"H0CRM1"	Q 662.0	BOOL	// [H0IM2.H0S21]: H0: COMANDO RECUO MOTOR M1
"H0CAM1"	Q 662.1	BOOL	// [H0IM2.H0S21]: H0: COMANDO AVANÇO MOTOR M1
"H0EAPLA"	Q 700.0	BOOL	// [H0DTS1]: H0: EV RETROCESO PILOTO A
"H0ERPLA"	Q 700.1	BOOL	// [H0DTS1]: H0: EV AVANCE PILOTO A
"H0EASRB"	Q 700.2	BOOL	// [H0DTS1]: H0: EV RETROCESO SERRAGE B
"H0ERSRB"	Q 700.3	BOOL	// [H0DTS1]: H0: EV AVANCE SERRAGE B
"H0EASRC"	Q 700.4	BOOL	// [H0DTS1]: H0: EV RETROCESO SERRAGE C
"H0ERSRC"	Q 700.5	BOOL	// [H0DTS1]: H0: EV AVANCE SERRAGE C
"H0EASRD"	Q 700.6	BOOL	// [H0DTS1]: H0: EV RETROCESO SERRAGE D
"H0ERSRD"	Q 700.7	BOOL	// [H0DTS1]: H0: EV AVANCE SERRAGE D
"H0EASRE"	Q 701.0	BOOL	// [H0DTS1]: H0: EV RETROCESO SERRAGE E
"H0ERSRE"	Q 701.1	BOOL	// [H0DTS1]: H0: EV AVANCE SERRAGE E
"H0EASRF"	Q 701.2	BOOL	// [H0DTS1]: H0: EV RETROCESO SERRAGE F
"H0ERSRF"	Q 701.3	BOOL	// [H0DTS1]: H0: EV AVANCE SERRAGE F
"H0EAPLG"	Q 701.4	BOOL	// [H0DTS1]: H0: EV RETROCESO PILOTO G - TRABA MOT
"H0ERPLG"	Q 701.5	BOOL	// [H0DTS1]: H0: EV AVANCE PILOTO G - TRABA MOT
"H0EAPLH"	Q 701.6	BOOL	// [H0DTS1]: H0: EV RETROCESO PILOTO H
"H0ERPLH"	Q 701.7	BOOL	// [H0DTS1]: H0: EV AVANCE PILOTO H
"H0EAPLI"	Q 702.0	BOOL	// [H0DTS1]: H0: EV Avance PILOTO I
"H0ERPLI"	Q 702.1	BOOL	// [H0DTS1]: H0: EV Retroceso PILOTO I
"Z2RCM"	Q 800.7	BOOL	// [Z2ZB.M05]: Z2 GROUND CONTROL RELAY
"Z2RSC1"	Q 815.0	BOOL	// [Z2ZB.M09]: RELAY SAFETY COMMON 1 (AU)
"Z2RES"	Q 815.1	BOOL	// [Z2ZB.M09]: RELAY SAFETY COMMON 2 (ES)
"Z2RFZ"	Q 815.2	BOOL	// [Z2ZB.M09]: RELAY SAFETY COMMON 3 (RFZ)
"Z2RSC4"	Q 815.3	BOOL	// [Z2ZB.M09]: RELAY SAFETY COMMON 4 (SC4)
"B1OP1VAT"	Q 821.0	BOOL	// B1 Lampara autorizacion de trabajo
"B1OP1VIT"	Q 821.1	BOOL	// B1 Lampara de prohibicion de trabajo
"B1OP1VDF"	Q 821.2	BOOL	// B1 Lampara de defecto
"B0RFRO1"	Q 841.0	BOOL	// [B0SB.M11]: B0 SAFETY COMMON 3 (FRO1)
"B0RFRO2"	Q 841.1	BOOL	// [B0SB.M11]: B0 SAFETY COMMON 4 (FRO2)
"B0RFRO3"	Q 841.2	BOOL	// [B0SB.M11]: B0 SAFETY COMMON 5 (FRO3)
"C1OP1VAT"	Q 851.0	BOOL	// C1 Lampara autorizacion de trabajo
"C1OP1VIT"	Q 851.1	BOOL	// C1 Lampara de prohibicion de trabajo
"C1OP1VDF"	Q 851.2	BOOL	// C1 Lampara de defecto
"C0RFRO1"	Q 871.0	BOOL	// [C0SB.M11]: C0 SAFETY COMMON 3 (C0SOP)
"C0RFRO2"	Q 871.1	BOOL	// [C0SB.M11]: C0 SAFETY COMMON 4 (C0)
"C0RFRO3"	Q 871.2	BOOL	// [C0SB.M11]: C0 SAFETY COMMON 5 (C0)
"E1OP1VAT"	Q 881.0	BOOL	// E1 Lampara autorizacion de trabajo
"E1OP1VIT"	Q 881.1	BOOL	// E1 Lampara de prohibicion de trabajo
"E1OP1VDF"	Q 881.2	BOOL	// E1 Lampara de defecto
"E0RFRO1"	Q 901.0	BOOL	// [E0SB.M11]: E0 SAFETY COMMON 3 ( E0SOP)
"E0RFRO2"	Q 901.1	BOOL	// [E0SB.M11]: E0 SAFETY COMMON 4 ( E0)
"E0RFRO3"	Q 901.2	BOOL	// [E0SB.M11]: E0 SAFETY COMMON 5 ( E0)
"G1OP1VAT"	Q 911.0	BOOL	// B1 Lampara autorizacion de trabajo
"G1OP1VIT"	Q 911.1	BOOL	// B1 Lampara de prohibicion de trabajo
"G1OP1VDF"	Q 911.2	BOOL	// B1 Lampara de defecto
"G0RFRO1"	Q 931.0	BOOL	// [G0SB.M11]: G0 SAFETY COMMON 3 (G0SOP)
"G0RFRO2"	Q 931.1	BOOL	// [G0SB.M11]: G0 SAFETY COMMON 4 (G0)
"G0RFRO3"	Q 931.2	BOOL	// [G0SB.M11]: G0 SAFETY COMMON 5 (G0)
"J1OP1VAT"	Q 940.0	BOOL	// J1 Lampara autorizacion de trabajo
"J1OP1VIT"	Q 940.1	BOOL	// J1 Lampara de prohibicion de trabajo
"J1OP1VDF"	Q 940.2	BOOL	// J1 Lampara de defecto
"B0EAPL1"	Q 950.0	BOOL	// [B0DTS1]: B0: EV AVANCE PL1
"B0ERPL1"	Q 950.1	BOOL	// [B0DTS1]: B0: EV RETROCESO PL1
"B0EASR2"	Q 950.2	BOOL	// [B0DTS1]: B0: EV AVANCE SR2
"B0ERSR2"	Q 950.3	BOOL	// [B0DTS1]: B0: EV RETROCESO SR2
"B0EASR3"	Q 950.4	BOOL	// [B0DTS1]: B0: EV AVANCE SR3
"B0ERSR3"	Q 950.5	BOOL	// [B0DTS1]: B0: EV RETROCESO SR3
"C0EAPL1"	Q 960.0	BOOL	// [C0DTS1]: C0: EV AVANCE PL1
"C0ERPL1"	Q 960.1	BOOL	// [C0DTS1]: C0: EV RETROCESO PL1
"C0EASR2"	Q 961.2	BOOL	// [C0DTS1]: C0: EV AVANCE SR2
"C0ERSR2"	Q 961.3	BOOL	// [C0DTS1]: C0: EV RETROCESO SR2
"C0EASR3"	Q 961.4	BOOL	// [C0DTS1]: C0: EV AVANCE SR3
"C0ERSR3"	Q 961.5	BOOL	// [C0DTS1]: C0: EV RETROCESO SR3
"E0EASR1"	Q 1040.0	BOOL	// [E0TDS1]: E0: EV AVANCE SR1
"E0ERSR1"	Q 1040.1	BOOL	// [E0TDS1]: E0: EV RETROCESO SR1
"E0EASR2"	Q 1040.2	BOOL	// [E0TDS1]: E0: EV AVANCE SR2
"E0ERSR2"	Q 1040.3	BOOL	// [E0TDS1]: E0: EV RETROCESO SR2
"E0EASR3"	Q 1040.4	BOOL	// [E0TDS1]: E0: EV AVANCE SR3
"E0ERSR3"	Q 1040.5	BOOL	// [E0TDS1]: E0: EV RETROCESO SR3
"E0EAVU4"	Q 1040.6	BOOL	// [E0TDS1]: E0: EV AVANCE VU4
"E0ERVU4"	Q 1040.7	BOOL	// [E0TDS1]: E0: EV RETROCESO VU4
"E0EAVU5"	Q 1041.0	BOOL	// [E0TDS1]: E0: EV AVANCE VU5
"E0ERVU5"	Q 1041.1	BOOL	// [E0TDS1]: E0: EV RETROCESO VU5
"E0EASR6"	Q 1041.2	BOOL	// [E0TDS1]: E0: EV AVANCE SR6
"E0ERSR6"	Q 1041.3	BOOL	// [E0TDS1]: E0: EV RETROCESO SR6
"G0EASR1"	Q 1060.0	BOOL	// [G0TDS1]: G0: EV AVANCE SR1
"G0ERSR1"	Q 1060.1	BOOL	// [G0TDS1]: G0: EV RETROCESO SR1
"G0EASR2"	Q 1060.2	BOOL	// [G0TDS1]: G0: EV AVANCE SR2
"G0ERSR2"	Q 1060.3	BOOL	// [G0TDS1]: G0: EV RETROCESO SR2
"G0EASR3"	Q 1060.4	BOOL	// [G0TDS1]: G0: EV AVANCE SR3
"G0ERSR3"	Q 1060.5	BOOL	// [G0TDS1]: G0: EV RETROCESO SR3
"TP"	SFB 3	SFB 3	// GENERATE A PULSE
"TON"	SFB 4	SFB 4	// GENERATE AN ON DELAY
"TOF"	SFB 5	SFB 5	// GENERATE AN OFF DELAY
"RDREC"	SFB 52	SFB 52	// READ A PROCESS DATA RECORD
"WRREC"	SFB 53	SFB 53	// WRITE A PROCESS DATA RECORD
"RALRM"	SFB 54	SFB 54	// Receive Alarm Data
"SET_CLK"	SFC 0	SFC 0	// SET SYSTEM CLOCK
"READ_CLK"	SFC 1	SFC 1	// READ SYSTEM CLOCK
"RD_SINFO"	SFC 6	SFC 6	// READ OB START INFORMATION
"D_ACT_DP"	SFC 12	SFC 12	// DEACTIVATING AND ACTIVATING DP SLAVES
"DPRD_DAT"	SFC 14	SFC 14	// READ CONSISTENT DATA OF A STANDARD DP SLAVE
"DPWR_DAT"	SFC 15	SFC 15	// WRITE CONSISTENT DATA TO A STANDARD DP SLAVE
"BLKMOV"	SFC 20	SFC 20	// COPY VARIABLES
"FILL"	SFC 21	SFC 21	// INITIALIZE A MEMORY AREA
"TEST_DB"	SFC 24	SFC 24	// TEST DATA BLOCK
"DIS_AIRT"	SFC 41	SFC 41	// DELAY THE HIGHER PRIORITY INTERRUPTS AND ASYNCHRONOUS ERRORS
"EN_AIRT"	SFC 42	SFC 42	// ENABLE HIGHER PRIORITY INTERRUPTS AND ASYNCHRONOUS ERRORS
"STP"	SFC 46	SFC 46	// CHANGE THE CPU TO STOP
"RDSYSST"	SFC 51	SFC 51	// READ A SYSTEM STATUS LIST OR PARTIAL LIST
"WR_REC"	SFC 58	SFC 58	// WRITE DATA RECORD
"RD_REC"	SFC 59	SFC 59	// READ A DATA RECORD
"TIME_TCK"	SFC 64	SFC 64	// READ THE SYSTEM TIME
"GEO_LOG"	SFC 70	SFC 70	// DETERMINE LOGICAL ADDRESS
"READ_DBL"	SFC 83	SFC 83	// READ DATA BLOCK OUT OF LOAD MEMORY
"WRIT_DBL"	SFC 84	SFC 84	// WRITE DATA BLOCK IN LOAD MEMORY
"DEL_SI"	SFC 106	SFC 106	// Deleting Dynamically Assigned System Instances
"ALARM_DQ"	SFC 107	SFC 107	// Creating Acknowledgeable Block-related Message
"ALARM_D"	SFC 108	SFC 108	// Creating Acknowledged Block-related Message
"LIEN_SEC"	UDT 1507	UDT 1507	// TABLE COMMUNE AUX BF_ZONE_PORTE1, BF_ZONE_RSEC1, BF_ZONE_MODE_IHM, BF_ZONE_AIR
"MOT_FONC_DPL"	UDT 1866	UDT 1866
"LIEN_PUP"	UDT 1988	UDT 1988	// Gestion des Modes et des pupitres de cde manu de la  zone (BF_ZONE_MODE_IHM)
"LIEN_ILOT"	UDT 2004	UDT 2004	// INFO CONTROL LINKED TO THE FACILITY (BF_ILOT)
"MOT_FONC_MP"	UDT 2041	UDT 2041	// INFO CONTROL OF A MOVEMENT (BF_MOUVMP1)
"MOT_FONC"	UDT 2042	UDT 2042
"VAT_SIPTOL"	VAT 1	
"VAT_TALOA0"	VAT 2	
"VAT_BASE DE DADOS"	VAT 3	
"Z1T_TEMPOS"	VAT 4	
"Z2T_TEMPOS"	VAT 5	
"VAT_6"	VAT 6	
"acompanhamento zona 8"	VAT 7		// teste tucker
"TOMAS"	VAT 8	
"W0"	VAT 9	
"VAT_Z1_BOT_EMER"	VAT 10	
"VAT_Z2_BOT_EMER"	VAT 11		// BOTAO_DE_EMERGENCIA
"VAT_Z1_VALIDAÇÃO"	VAT 12	
"VAT_CDIV_2"	VAT 13	
"VAT_Z2_VALIDAÇÃO"	VAT 14	
"ELEV_CARREGAMENTO"	VAT 15	
"ELEV_DESCARREGAMENTO"	VAT 16	
"VAT_17"	VAT 17	
"TESTE_MODO_DEGR"	VAT 18	
"VAT_SIPTOL_TOM"	VAT 19	
"mostrar IIT"	VAT 20	
"tab_iit_2"	VAT 21	
"VAT_22"	VAT 22	
"afficher"	VAT 23	
"VAT_24"	VAT 24	
END_SYMBOL_TABLE
